(* IEC 61131-3 sources: Industry-PLC-LLM/data/PLCBEAD_repo/PLCBEAD_PLCEmbed-main/PLC-BEAD/Source/OpenPLCv2 (part 12) *)

(* ---- RES_NI.ST ---- *)
FUNCTION RES_NI:REAL

	VAR_INPUT
		T :	REAL;
		R0 :	REAL;
	END_VAR

	VAR
		T2 :	REAL;
	END_VAR

	T2 := T*T;
	Res_NI := R0 + 0.5485*T + 0.665E-3*T2 + 2.805E-9*T2*T2;

END_FUNCTION

PROGRAM program0

	VAR
		T :	REAL;
		R0 :	REAL;

		OUT :	REAL;
	END_VAR
	OUT := RES_NI(T, R0);

END_PROGRAM

CONFIGURATION Config0

	RESOURCE Res0 ON PLC
		TASK task0(INTERVAL := T#20ms,PRIORITY := 0);
		PROGRAM instance0 WITH task0 : program0;
	END_RESOURCE

END_CONFIGURATION

(* ---- RES_NTC.ST ---- *)
FUNCTION RES_NTC:REAL

	VAR_INPUT
		T :	REAL;
		RN :	REAL;
		B :	REAL;
	END_VAR

	RES_NTC := RN * EXP(B * (1.0 / (T+273.15) - 0.00335401643468053));

END_FUNCTION

PROGRAM program0

	VAR
		T :	REAL;
		RN :	REAL;
		B :	REAL;

		OUT :	REAL;
	END_VAR
		OUT := RES_NTC(T, RN, B);

END_PROGRAM

CONFIGURATION Config0

	RESOURCE Res0 ON PLC
		TASK task0(INTERVAL := T#20ms,PRIORITY := 0);
		PROGRAM instance0 WITH task0 : program0;
	END_RESOURCE

END_CONFIGURATION

(* ---- RES_PT.ST ---- *)
FUNCTION RES_PT:REAL
	VAR_INPUT
		T :	REAL;
		R0 :	REAL;
	END_VAR

	VAR
		T2 :	REAL;
	END_VAR

	T2 := T * T;

	IF T >= 0.0 THEN
		RES_PT := R0 * ( 1.0 + 3.90802E-3 * T + -5.802E-7 * T2);
	ELSE
		RES_PT := R0 * ( 1.0 + 3.90802E-3 * T + -5.802E-7 * T2 + -4.27350E-12 * (T - 100.0) * T2 * T);
	END_IF;

END_FUNCTION

PROGRAM program0
  	VAR
		T :	REAL;
		R0 : REAL;
		CEIL5_OUT : REAL;
  	END_VAR

  	CEIL5_OUT := RES_PT(T, R0);
END_PROGRAM

CONFIGURATION Config0
	RESOURCE Res0 ON PLC
		TASK task0(INTERVAL := T#20ms,PRIORITY := 0);
		PROGRAM instance0 WITH task0 : program0;
	END_RESOURCE
END_CONFIGURATION

(* ---- RES_SI.ST ---- *)
FUNCTION RES_SI:REAL

	VAR_INPUT
		T :	REAL;
		_RS :	REAL;
		TS :	REAL;
	END_VAR

	VAR
		TX :	REAL;
	END_VAR

	TX := T - TS;
	RES_SI := _RS * ( 1.0 + 7.64E-3 * TX + 1.66E-5 * TX * TX);

END_FUNCTION

PROGRAM program0

	VAR
		T :	REAL;
		_RS :	REAL;
		TS :	REAL;

		OUT :	REAL;
	END_VAR
		OUT := RES_SI(T, _RS, TS);

END_PROGRAM

CONFIGURATION Config0

	RESOURCE Res0 ON PLC
		TASK task0(INTERVAL := T#20ms,PRIORITY := 0);
		PROGRAM instance0 WITH task0 : program0;
	END_RESOURCE

END_CONFIGURATION

(* ---- REVERSE.ST ---- *)
FUNCTION REVERSE:BYTE
VAR_INPUT
	IN :	BYTE;
END_VAR

reverse := SHL(in,7) OR SHR(in,7) OR (ROR(in,3) AND BYTE#2#01000100) OR (ROL(in,3) AND BYTE#2#00100010)
	OR (SHL(in,1) AND BYTE#2#00010000) OR (SHR(in,1) AND BYTE#2#00001000);

END_FUNCTION

PROGRAM program0
  VAR
    LocalVar0 : BYTE;
	LocalOUT  : BYTE;
  END_VAR
  	LocalOUT := REVERSE(LocalVar0);
END_PROGRAM

CONFIGURATION Config0
  RESOURCE Res0 ON PLC
    TASK task0(INTERVAL := T#20ms,PRIORITY := 0);
    PROGRAM instance0 WITH task0 : program0;
  END_RESOURCE
END_CONFIGURATION

(* ---- RND.ST ---- *)
FUNCTION CEIL:INT

	VAR_INPUT
		X :	REAL;
	END_VAR

	CEIL := REAL_TO_INT(x);
	IF INT_TO_REAL(CEIL) < X THEN
			CEIL := CEIL + 1;
	END_IF;

END_FUNCTION

FUNCTION BIT_OF_DWORD : BOOL

	VAR_INPUT
		IN : DWORD;
		N : INT;
	END_VAR

	BIT_OF_DWORD := (SHR(in,N) AND 16#00000001) > 0;

END_FUNCTION

FUNCTION EXPN:REAL

	VAR_INPUT
		X :	REAL;
		N :	INT;
	END_VAR

	VAR
		N_word :	WORD;
		X_tmp :	REAL;
		sign :	BOOL;
	END_VAR

	N_word := INT_TO_WORD(N);
	X_tmp := X;
	sign := BIT_OF_DWORD(WORD_TO_DWORD(N_word),15);
	N_word := INT_TO_WORD(ABS(N));
	IF BIT_OF_DWORD(WORD_TO_DWORD(N_word),0) THEN expn := X_tmp; ELSE expn := 1.0; END_IF;    (* N_word.X0 *)
	N_word := SHR(N_word,1);
	WHILE N_word > WORD#0 DO
		X_tmp := X_tmp * X_tmp;
		IF BIT_OF_DWORD(WORD_TO_DWORD(N_word),0) THEN expn := expn * X_tmp; END_IF;       (* N_word.X0 *)
		N_word := SHR(N_word,1);
	END_WHILE;
	IF sign THEN EXPN := 1.0 / EXPN; END_IF;

END_FUNCTION

FUNCTION _REAL_TO_DINT:DINT
	VAR_INPUT
		X :	REAL;
	END_VAR

	IF REAL_TO_DINT(0.5) = DINT#1 THEN
		_REAL_TO_DINT := REAL_TO_DINT(x);
		RETURN;
	END_IF;

	IF X > 0.0 THEN
		_REAL_TO_DINT := REAL_TO_DINT(x+0.5);
	ELSIF X < 0.0 THEN
		_REAL_TO_DINT := REAL_TO_DINT(x-0.5);
	ELSE
		_REAL_TO_DINT := DINT#0;
	END_IF;
END_FUNCTION

FUNCTION RND:REAL

	VAR_INPUT
		X :	REAL;
		N :	INT;
	END_VAR

	VAR
		M :	REAL;
	END_VAR

	IF X = 0.0 THEN
		RND := 0.0;
	ELSE
		M := EXPN(10.0,N - CEIL(LOG(ABS(X))));
		RND := DINT_TO_REAL(_REAL_TO_DINT(X * M)) / M;
	END_IF;

END_FUNCTION

PROGRAM program0
	VAR
		IN : REAL;
		N :	INT;
		X :	REAL;
	END_VAR
		X := RND(IN, N);
END_PROGRAM

CONFIGURATION Config0

	RESOURCE Res0 ON PLC
		TASK task0(INTERVAL := T#20ms,PRIORITY := 0);
		PROGRAM instance0 WITH task0 : program0;
	END_RESOURCE

END_CONFIGURATION

(* ---- ROUND.ST ---- *)
FUNCTION _REAL_TO_DINT:DINT
	VAR_INPUT
		X :	REAL;
	END_VAR

	IF REAL_TO_DINT(0.5) = DINT#1 THEN
		_REAL_TO_DINT := REAL_TO_DINT(x);
		RETURN;
	END_IF;

	IF X > 0.0 THEN
		_REAL_TO_DINT := REAL_TO_DINT(x+0.5);
	ELSIF X < 0.0 THEN
		_REAL_TO_DINT := REAL_TO_DINT(x-0.5);
	ELSE
		_REAL_TO_DINT := DINT#0;
	END_IF;
END_FUNCTION

FUNCTION ROUND:REAL

	VAR_INPUT
		IN :	REAL;
		N :	INT;
	END_VAR

	VAR
		X :	REAL;
	END_VAR

	IF N < 4 THEN
		IF N < 2 THEN
			IF N = 0 THEN X := 1.0; ELSE X := 10.0; END_IF;
		ELSE
			IF N = 2 THEN X := 100.0; ELSE X := 1000.0; END_IF;
		END_IF;
	ELSE
		IF N < 6 THEN
			IF N = 4 THEN X := 10000.0; ELSE X := 100000.0; END_IF;
		ELSE
			IF N = 6 THEN X := 1000000.0; ELSE X := 10000000.0; END_IF;
		END_IF;
	END_IF;

	ROUND := DINT_TO_REAL(_REAL_TO_DINT(in * X)) / X;

END_FUNCTION

PROGRAM program0
	VAR
		IN : REAL;
		N :	INT;
		X :	REAL;
	END_VAR
		X := ROUND(IN, N);
END_PROGRAM

CONFIGURATION Config0

	RESOURCE Res0 ON PLC
		TASK task0(INTERVAL := T#20ms,PRIORITY := 0);
		PROGRAM instance0 WITH task0 : program0;
	END_RESOURCE

END_CONFIGURATION

(* ---- SCALE.ST ---- *)
FUNCTION SCALE:REAL

	VAR_INPUT
		X :	REAL;
		K :	REAL;
		O :	REAL;
		MX :	REAL;
		MN :	REAL;
	END_VAR

	SCALE := LIMIT(MN, X * K + O, MX);

END_FUNCTION

PROGRAM program0
  VAR
    X :	REAL;
	K :	REAL;
	O :	REAL;
	MX :	REAL;
	MN :	REAL;
    CEIL5_OUT : REAL;
  END_VAR

  CEIL5_OUT := SCALE(X, K, O, MX, MN);
END_PROGRAM

CONFIGURATION Config0

  RESOURCE Res0 ON PLC
    TASK task0(INTERVAL := T#20ms,PRIORITY := 0);
    PROGRAM instance0 WITH task0 : program0;
  END_RESOURCE
END_CONFIGURATION

(* ---- SCALE_B.ST ---- *)
FUNCTION _BYTE_TO_REAL:REAL
	VAR_INPUT
		IN :	BYTE;
	END_VAR

	_BYTE_TO_REAL := USINT_TO_REAL(BYTE_TO_USINT(IN));
END_FUNCTION

FUNCTION SCALE_B:REAL

	VAR_INPUT
		X :	BYTE;
		I_LO :	BYTE;
		I_HI :	BYTE;
		O_LO :	REAL;
		O_HI :	REAL;
	END_VAR

	IF I_HI = I_LO THEN
		SCALE_B := O_LO;
	ELSE
		SCALE_B := (O_HI - O_LO) / USINT_TO_REAL(BYTE_TO_USINT(I_HI) - BYTE_TO_USINT(I_LO)) * _BYTE_TO_REAL(LIMIT(I_LO,X,I_HI));
	END_IF;

END_FUNCTION

PROGRAM program0
  VAR
	X :	BYTE;
	I_LO :	BYTE;
	I_HI :	BYTE;
	O_LO :	REAL;
	O_HI :	REAL;
	CEIL5_OUT : REAL;
  END_VAR

  CEIL5_OUT := SCALE_B(X, I_LO, I_HI, O_LO, O_HI);

END_PROGRAM

CONFIGURATION Config0

  RESOURCE Res0 ON PLC
    TASK task0(INTERVAL := T#20ms,PRIORITY := 0);
    PROGRAM instance0 WITH task0 : program0;
  END_RESOURCE
END_CONFIGURATION

(* ---- SCALE_B2.ST ---- *)
FUNCTION _BYTE_TO_REAL:REAL
	VAR_INPUT
		IN :	BYTE;
	END_VAR

	_BYTE_TO_REAL := USINT_TO_REAL(BYTE_TO_USINT(IN));
END_FUNCTION

FUNCTION SCALE_B2:REAL
	VAR_INPUT
		IN1 :	BYTE;
		IN2 :	BYTE;
		K :	REAL;
		O :	REAL;
		IN1_MIN :	REAL;
		IN1_MAX :	REAL;
		IN2_MIN :	REAL;
		IN2_MAX :	REAL;
	END_VAR

	SCALE_B2 := 	(((in1_max - in1_min)* _BYTE_TO_REAL(in1) + (in2_max - in2_min)* _BYTE_TO_REAL(in2)) * 0.003921569 + in1_min + in2_min) * K + O;

END_FUNCTION

PROGRAM program0
  VAR
	IN1 :	BYTE;
	IN2 :	BYTE;
	K :	REAL;
	O :	REAL;
	IN1_MIN :	REAL;
	IN1_MAX :	REAL;
	IN2_MIN :	REAL;
	IN2_MAX :	REAL;
	CEIL5_OUT : REAL;
  END_VAR

  CEIL5_OUT := SCALE_B2(IN1, IN2, K, O, IN1_MIN, IN1_MAX, IN2_MIN, IN2_MAX);

END_PROGRAM

CONFIGURATION Config0

  RESOURCE Res0 ON PLC
    TASK task0(INTERVAL := T#20ms,PRIORITY := 0);
    PROGRAM instance0 WITH task0 : program0;
  END_RESOURCE
END_CONFIGURATION

(* ---- SCALE_B4.ST ---- *)
FUNCTION _BYTE_TO_REAL:REAL
	VAR_INPUT
		IN :	BYTE;
	END_VAR

	_BYTE_TO_REAL := USINT_TO_REAL(BYTE_TO_USINT(IN));
END_FUNCTION

FUNCTION SCALE_B4:REAL

	VAR_INPUT
		IN1 :	BYTE;
		IN2 :	BYTE;
		IN3 :	BYTE;
		IN4 :	BYTE;
		K :	REAL;
		O :	REAL;
		IN1_MIN :	REAL;
		IN1_MAX :	REAL;
		IN2_MIN :	REAL;
		IN2_MAX :	REAL;
		IN3_MIN :	REAL;
		IN3_MAX :	REAL;
		IN4_MIN :	REAL;
		IN4_MAX :	REAL;
	END_VAR

	SCALE_B4 := 	(((in1_max - in1_min)* _BYTE_TO_REAL(in1) + (in2_max - in2_min)* _BYTE_TO_REAL(in2) + (in3_max - in3_min)* _BYTE_TO_REAL(in3) + (in4_max - in4_min)* _BYTE_TO_REAL(in4))* 0.003921569 + in1_min + in2_min + in3_min + in4_min) * K + O;

END_FUNCTION

PROGRAM program0
  VAR
	IN1 :	BYTE;
	IN2 :	BYTE;
	IN3 :	BYTE;
	IN4 :	BYTE;
	K :	REAL;
	O :	REAL;
	IN1_MIN :	REAL;
	IN1_MAX :	REAL;
	IN2_MIN :	REAL;
	IN2_MAX :	REAL;
	IN3_MIN :	REAL;
	IN3_MAX :	REAL;
	IN4_MIN :	REAL;
	IN4_MAX :	REAL;
	CEIL5_OUT : REAL;
  END_VAR

  CEIL5_OUT := SCALE_B4(IN1, IN2, IN3, IN4, K, O, IN1_MIN, IN1_MAX, IN2_MIN, IN2_MAX, IN3_MIN, IN3_MAX, IN4_MIN, IN4_MAX);

END_PROGRAM

CONFIGURATION Config0

  RESOURCE Res0 ON PLC
    TASK task0(INTERVAL := T#20ms,PRIORITY := 0);
    PROGRAM instance0 WITH task0 : program0;
  END_RESOURCE
END_CONFIGURATION

(* ---- SCALE_B8.ST ---- *)
FUNCTION _BYTE_TO_REAL:REAL
	VAR_INPUT
		IN :	BYTE;
	END_VAR

	_BYTE_TO_REAL := USINT_TO_REAL(BYTE_TO_USINT(IN));
END_FUNCTION

FUNCTION SCALE_B8:REAL
	VAR_INPUT
		IN1 :	BYTE;
		IN2 :	BYTE;
		IN3 :	BYTE;
		IN4 :	BYTE;
		IN5 :	BYTE;
		IN6 :	BYTE;
		IN7 :	BYTE;
		IN8 :	BYTE;
		K :	REAL;
		O :	REAL;
		IN1_MIN :	REAL;
		IN1_MAX :	REAL;
		IN2_MIN :	REAL;
		IN2_MAX :	REAL;
		IN3_MIN :	REAL;
		IN3_MAX :	REAL;
		IN4_MIN :	REAL;
		IN4_MAX :	REAL;
		IN5_MIN :	REAL;
		IN5_MAX :	REAL;
		IN6_MIN :	REAL;
		IN6_MAX :	REAL;
		IN7_MIN :	REAL;
		IN7_MAX :	REAL;
		IN8_MIN :	REAL;
		IN8_MAX :	REAL;
	END_VAR

	SCALE_B8 := 	(((in1_max - in1_min)* _BYTE_TO_REAL(in1) + (in2_max - in2_min)* _BYTE_TO_REAL(in2) + (in3_max - in3_min)* _BYTE_TO_REAL(in3) + (in4_max - in4_min)* _BYTE_TO_REAL(in4) +
					(in5_max - in5_min)* _BYTE_TO_REAL(in5) + (in6_max - in6_min)* _BYTE_TO_REAL(in6) + (in7_max - in7_min)* _BYTE_TO_REAL(in7) + (in8_max - in8_min)* _BYTE_TO_REAL(in8)) * 0.003921569
					+ in1_min + in2_min + in3_min + in4_min + in5_min + in6_min + in7_min + in8_min) * K + O;

END_FUNCTION

PROGRAM program0
  	VAR
		IN1 :	BYTE;
		IN2 :	BYTE;
		IN3 :	BYTE;
		IN4 :	BYTE;
		IN5 :	BYTE;
		IN6 :	BYTE;
		IN7 :	BYTE;
		IN8 :	BYTE;
		K :	REAL;
		O :	REAL;
		IN1_MIN :	REAL;
		IN1_MAX :	REAL;
		IN2_MIN :	REAL;
		IN2_MAX :	REAL;
		IN3_MIN :	REAL;
		IN3_MAX :	REAL;
		IN4_MIN :	REAL;
		IN4_MAX :	REAL;
		IN5_MIN :	REAL;
		IN5_MAX :	REAL;
		IN6_MIN :	REAL;
		IN6_MAX :	REAL;
		IN7_MIN :	REAL;
		IN7_MAX :	REAL;
		IN8_MIN :	REAL;
		IN8_MAX :	REAL;
		CEIL5_OUT : REAL;
  	END_VAR

  	CEIL5_OUT := SCALE_B8(IN1, IN2, IN3, IN4, IN5, IN6, IN7, IN8, K, O, IN1_MIN, IN1_MAX, IN2_MIN, IN2_MAX, IN3_MIN, IN3_MAX, IN4_MIN, IN4_MAX, IN5_MIN, IN5_MAX, IN6_MIN, IN6_MAX, IN7_MIN, IN7_MAX, IN8_MIN, IN8_MAX);

	END_PROGRAM

CONFIGURATION Config0

	RESOURCE Res0 ON PLC
		TASK task0(INTERVAL := T#20ms,PRIORITY := 0);
		PROGRAM instance0 WITH task0 : program0;
	END_RESOURCE

END_CONFIGURATION

(* ---- SCALE_D.ST ---- *)
FUNCTION SCALE_D:REAL
	VAR_INPUT
		X :	DWORD;
		I_LO :	DWORD;
		I_HI :	DWORD;
		O_LO :	REAL;
		O_HI :	REAL;
	END_VAR
	IF I_HI = I_LO THEN
		SCALE_D := O_LO;
	ELSE
		SCALE_D := (O_HI - O_LO) / UDINT_TO_REAL(DWORD_TO_UDINT(I_HI) - DWORD_TO_UDINT(I_LO)) * UDINT_TO_REAL(LIMIT(DWORD_TO_UDINT(I_LO),DWORD_TO_UDINT(X),DWORD_TO_UDINT(I_HI)) - DWORD_TO_UDINT(I_LO)) + O_LO;
	END_IF;
END_FUNCTION

PROGRAM program0
  VAR
		X :	DWORD;
		I_LO :	DWORD;
		I_HI :	DWORD;
		O_LO :	REAL;
		O_HI :	REAL;
		CEIL5_OUT : REAL;
  END_VAR

  CEIL5_OUT := SCALE_D(X, I_LO, I_HI, O_LO, O_HI);
END_PROGRAM

CONFIGURATION Config0

  RESOURCE Res0 ON PLC
    TASK task0(INTERVAL := T#20ms,PRIORITY := 0);
    PROGRAM instance0 WITH task0 : program0;
  END_RESOURCE
END_CONFIGURATION

(* ---- SCALE_R.ST ---- *)
FUNCTION SCALE_R:REAL
	VAR_INPUT
		X :	REAL;
		I_LO :	REAL;
		I_HI :	REAL;
		O_LO :	REAL;
		O_HI :	REAL;
	END_VAR

	IF I_LO = I_HI THEN
		SCALE_R := O_LO;
	ELSE
		SCALE_R := (O_HI - O_LO) / (I_HI - I_LO) * (LIMIT(I_LO, X, I_HI) - I_LO) + O_LO;
	END_IF;

END_FUNCTION

PROGRAM program0

  	VAR
		X :	REAL;
		I_LO :	REAL;
		I_HI :	REAL;
		O_LO :	REAL;
		O_HI :	REAL;
		CEIL5_OUT : REAL;
  	END_VAR

  	CEIL5_OUT := SCALE_R(X, I_LO, I_HI, O_LO, O_HI);
END_PROGRAM

CONFIGURATION Config0

	RESOURCE Res0 ON PLC
		TASK task0(INTERVAL := T#20ms,PRIORITY := 0);
		PROGRAM instance0 WITH task0 : program0;
	END_RESOURCE

END_CONFIGURATION

(* ---- SCALE_X2.ST ---- *)
FUNCTION SCALE_X2:REAL
	VAR_INPUT
		IN1 :	BOOL;
		IN2 :	BOOL;
		K :	REAL;
		O :	REAL;
		IN1_MIN :	REAL;(*Standard = 0*)
		IN1_MAX :	REAL;(*Standard = 1000*)
		IN2_MIN :	REAL;(*Standard = 0*)
		IN2_MAX :	REAL;(*Standard = 1000*)
	END_VAR

	SCALE_X2 := (SEL(IN1,IN1_MIN, IN1_MAX)+ SEL(IN2,IN2_MIN, IN2_MAX))* k + o;

END_FUNCTION

PROGRAM program0

  	VAR
		IN1 :	BOOL;
		IN2 :	BOOL;
		K :	REAL;
		O :	REAL;
		IN1_MIN :	REAL;(*Standard = 0*)
		IN1_MAX :	REAL;(*Standard = 1000*)
		IN2_MIN :	REAL;(*Standard = 0*)
		IN2_MAX :	REAL;(*Standard = 1000*)
		CEIL5_OUT : REAL;
  	END_VAR

  	CEIL5_OUT := SCALE_X2(IN1, IN2, K, O, IN1_MIN, IN1_MAX, IN2_MIN, IN2_MAX);
END_PROGRAM

CONFIGURATION Config0

	RESOURCE Res0 ON PLC
		TASK task0(INTERVAL := T#20ms,PRIORITY := 0);
		PROGRAM instance0 WITH task0 : program0;
	END_RESOURCE

END_CONFIGURATION

(* ---- SCALE_X4.ST ---- *)
FUNCTION SCALE_X4:REAL
	VAR_INPUT
		IN1 :	BOOL;
		IN2 :	BOOL;
		IN3 :	BOOL;
		IN4 :	BOOL;
		K :	REAL;
		O :	REAL;
		IN1_MIN :	REAL;
		IN1_MAX :	REAL;
		IN2_MIN :	REAL;
		IN2_MAX :	REAL;
		IN3_MIN :	REAL;
		IN3_MAX :	REAL;
		IN4_MIN :	REAL;
		IN4_MAX :	REAL;
	END_VAR
	IF NOT in1 THEN scale_X4 := in1_min; ELSE scale_X4 := in1_max; END_IF;
	IF NOT in2 THEN scale_x4 := scale_x4 + in2_min; ELSE scale_x4 := scale_x4 + in2_max; END_IF;
	IF NOT in3 THEN scale_x4 := scale_x4 + in3_min; ELSE scale_x4 := scale_x4 + in3_max; END_IF;
	IF NOT in4 THEN scale_x4 := scale_x4 + in4_min; ELSE scale_x4 := scale_x4 + in4_max; END_IF;
	scale_X4 := scale_X4 * k + O;
	END_FUNCTION

PROGRAM program0

  	VAR
		IN1 :	BOOL;
		IN2 :	BOOL;
		IN3 :	BOOL;
		IN4 :	BOOL;
		K :	REAL;
		O :	REAL;
		IN1_MIN :	REAL;
		IN1_MAX :	REAL;
		IN2_MIN :	REAL;
		IN2_MAX :	REAL;
		IN3_MIN :	REAL;
		IN3_MAX :	REAL;
		IN4_MIN :	REAL;
		IN4_MAX :	REAL;
		CEIL5_OUT : REAL;
  	END_VAR

  	CEIL5_OUT := SCALE_X4(IN1, IN2, IN3, IN4, K, O, IN1_MIN, IN1_MAX, IN2_MIN, IN2_MAX, IN3_MIN, IN3_MAX, IN4_MIN, IN4_MAX);
END_PROGRAM

CONFIGURATION Config0

	RESOURCE Res0 ON PLC
		TASK task0(INTERVAL := T#20ms,PRIORITY := 0);
		PROGRAM instance0 WITH task0 : program0;
	END_RESOURCE

END_CONFIGURATION

(* ---- SCALE_X8.ST ---- *)
FUNCTION SCALE_X8:REAL

	VAR_INPUT
		IN1 :	BOOL;
		IN2 :	BOOL;
		IN3 :	BOOL;
		IN4 :	BOOL;
		IN5 :	BOOL;
		IN6 :	BOOL;
		IN7 :	BOOL;
		IN8 :	BOOL;
		K :	REAL;
		O :	REAL;
		IN1_MIN :	REAL;
		IN1_MAX :	REAL;
		IN2_MIN :	REAL;
		IN2_MAX :	REAL;
		IN3_MIN :	REAL;
		IN3_MAX :	REAL;
		IN4_MIN :	REAL;
		IN4_MAX :	REAL;
		IN5_MIN :	REAL;
		IN5_MAX :	REAL;
		IN6_MIN :	REAL;
		IN6_MAX :	REAL;
		IN7_MIN :	REAL;
		IN7_MAX :	REAL;
		IN8_MIN :	REAL;
		IN8_MAX :	REAL;
	END_VAR

	SCALE_X8 := (SEL(IN1,IN1_MIN, IN1_MAX)+ SEL(IN2,IN2_MIN, IN2_MAX)+SEL(IN3,IN3_MIN, IN3_MAX)+ SEL(IN4,IN4_MIN, IN4_MAX)
					+SEL(IN5,IN5_MIN, IN5_MAX)+ SEL(IN6,IN6_MIN, IN6_MAX)+SEL(IN7,IN7_MIN, IN7_MAX)+ SEL(IN8,IN8_MIN, IN8_MAX))*k + o;

END_FUNCTION

PROGRAM program0

  	VAR
		IN1 :	BOOL;
		IN2 :	BOOL;
		IN3 :	BOOL;
		IN4 :	BOOL;
		IN5 :	BOOL;
		IN6 :	BOOL;
		IN7 :	BOOL;
		IN8 :	BOOL;
		K :	REAL;
		O :	REAL;
		IN1_MIN :	REAL;
		IN1_MAX :	REAL;
		IN2_MIN :	REAL;
		IN2_MAX :	REAL;
		IN3_MIN :	REAL;
		IN3_MAX :	REAL;
		IN4_MIN :	REAL;
		IN4_MAX :	REAL;
		IN5_MIN :	REAL;
		IN5_MAX :	REAL;
		IN6_MIN :	REAL;
		IN6_MAX :	REAL;
		IN7_MIN :	REAL;
		IN7_MAX :	REAL;
		IN8_MIN :	REAL;
		IN8_MAX :	REAL;
		CEIL5_OUT : REAL;
  	END_VAR

  	CEIL5_OUT := SCALE_X8(IN1, IN2, IN3, IN4, IN5, IN6, IN7, IN8, K, O, IN1_MIN, IN1_MAX, IN2_MIN, IN2_MAX, IN3_MIN, IN3_MAX, IN4_MIN, IN4_MAX, IN5_MIN, IN5_MAX, IN6_MIN, IN6_MAX, IN7_MIN, IN7_MAX, IN8_MIN, IN8_MAX);
END_PROGRAM

CONFIGURATION Config0

	RESOURCE Res0 ON PLC
		TASK task0(INTERVAL := T#20ms,PRIORITY := 0);
		PROGRAM instance0 WITH task0 : program0;
	END_RESOURCE

END_CONFIGURATION

(* ---- SDD.ST ---- *)
FUNCTION SDD:REAL

	VAR_INPUT
		T :	REAL;
		ICE :	BOOL;
	END_VAR

	IF ice THEN
		SDD := 611.153 * EXP(22.4433 * T / (272.186 + T));
	ELSE
		SDD := 611.213 * EXP(17.5043 * T / (241.2 + T));
	END_IF;

END_FUNCTION

PROGRAM program0
  VAR
    T :	REAL;
	ICE :	BOOL;
    CEIL5_OUT : REAL;
  END_VAR

  CEIL5_OUT := SDD(T, ICE);
END_PROGRAM

CONFIGURATION Config0

  RESOURCE Res0 ON PLC
    TASK task0(INTERVAL := T#20ms,PRIORITY := 0);
    PROGRAM instance0 WITH task0 : program0;
  END_RESOURCE
END_CONFIGURATION

(* ---- SDD_NH3.ST ---- *)
FUNCTION SDD_NH3:REAL

	VAR_INPUT
		T :	REAL;
	END_VAR

	IF T < -33.65 THEN
		SDD_NH3 := EXP(7.3396511649 - ( 1166.7498002 / ( T + 192.37 )));
	ELSE
		SDD_NH3 := EXP(11.210964456 - ( 2564.9140075 / ( T + 262.741 )));
	END_IF;

END_FUNCTION

PROGRAM program0
  VAR
    T :	REAL;
    CEIL5_OUT : REAL;
  END_VAR

  CEIL5_OUT := SDD_NH3(T);
END_PROGRAM

CONFIGURATION Config0

  RESOURCE Res0 ON PLC
    TASK task0(INTERVAL := T#20ms,PRIORITY := 0);
    PROGRAM instance0 WITH task0 : program0;
  END_RESOURCE
END_CONFIGURATION

(* ---- SDT_NH3.ST ---- *)
FUNCTION SDT_NH3:REAL

	VAR_INPUT
		P :	REAL;
	END_VAR

	IF P < 1.0E-3 THEN
		SDT_NH3 := -110.0;
	ELSIF P < 1.0 THEN
		SDT_NH3 := 506.713 / (3.18757 - LOG(P)) - 192.37 ;
	ELSE
		SDT_NH3 := 1113.928 / (4.86886 - LOG(P)) - 262.71 ;
	END_IF;

END_FUNCTION

PROGRAM program0
  VAR
    P :	REAL;
    CEIL5_OUT : REAL;
  END_VAR

  CEIL5_OUT := SDT_NH3(P);
END_PROGRAM

CONFIGURATION Config0

  RESOURCE Res0 ON PLC
    TASK task0(INTERVAL := T#20ms,PRIORITY := 0);
    PROGRAM instance0 WITH task0 : program0;
  END_RESOURCE
END_CONFIGURATION

(* ---- SECOND.ST ---- *)
FUNCTION SECOND:REAL

	VAR_INPUT
		ITOD :	UDINT;
	END_VAR

	second := UDINT_TO_REAL(itod MOD UDINT#60000) / REAL#1000.00;

END_FUNCTION

PROGRAM program0
  VAR
    ITOD :	UDINT;
    CEIL5_OUT : REAL;
  END_VAR

  CEIL5_OUT := SECOND(ITOD);
END_PROGRAM

CONFIGURATION Config0

	RESOURCE Res0 ON PLC
		TASK task0(INTERVAL := T#20ms,PRIORITY := 0);
		PROGRAM instance0 WITH task0 : program0;
	END_RESOURCE

END_CONFIGURATION

(* ---- SECOND_OF_DT.ST ---- *)
FUNCTION SECOND_OF_DT:INT

	VAR_INPUT
		XDT :	UDINT;
	END_VAR

	SECOND_OF_DT := UDINT_TO_INT(XDT MOD UDINT#60);
END_FUNCTION

PROGRAM program0
  VAR
    LocalVar0 : UDINT;
	LocalOUT  : INT;
  END_VAR
  	LocalOUT := SECOND_OF_DT(LocalVar0);
END_PROGRAM

CONFIGURATION Config0
  RESOURCE Res0 ON PLC
    TASK task0(INTERVAL := T#20ms,PRIORITY := 0);
    PROGRAM instance0 WITH task0 : program0;
  END_RESOURCE
END_CONFIGURATION

(* ---- SECOND_TO_TIME.ST ---- *)
FUNCTION _REAL_TO_UDINT:UDINT
	VAR_INPUT
		X :	REAL;
	END_VAR

	IF REAL_TO_UDINT(0.5) = UDINT#1 THEN
		_REAL_TO_UDINT := REAL_TO_UDINT(x);
	ELSIF X > 0.0 THEN
		_REAL_TO_UDINT := REAL_TO_UDINT(x+0.5);
	ELSIF X < 0.0 THEN
		_REAL_TO_UDINT := REAL_TO_UDINT(x-0.5);
	ELSE
		_REAL_TO_UDINT := UDINT#0;
	END_IF;
END_FUNCTION

FUNCTION SECOND_TO_TIME:TIME

	VAR_INPUT
		IN :	REAL;
	END_VAR

	second_to_time := UDINT_TO_TIME(_REAL_TO_UDINT(IN * 1000.0));

END_FUNCTION

PROGRAM program0

	VAR
		IN :	REAL;
		CEIL5_OUT : TIME;
	END_VAR

	CEIL5_OUT := SECOND_TO_TIME(IN);

END_PROGRAM

CONFIGURATION Config0

	RESOURCE Res0 ON PLC
		TASK task0(INTERVAL := T#20ms,PRIORITY := 0);
		PROGRAM instance0 WITH task0 : program0;
	END_RESOURCE

END_CONFIGURATION

(* ---- SENSOR_INT.ST ---- *)
FUNCTION SENSOR_INT:REAL

	VAR_INPUT
		VOLTAGE :	REAL;
		CURRENT :	REAL;
		RP :	REAL;
		_RS :	REAL;
	END_VAR

	VAR
		RG :	REAL;
	END_VAR

	IF current <> 0.0 THEN
		RG := voltage / current;
		SENSOR_INT := RP * ( RG - _RS) / ( RP + _RS - RG);
	END_IF;

END_FUNCTION

PROGRAM program0

	VAR
		VOLTAGE :	REAL;
		CURRENT :	REAL;
		RP :	REAL;
		_RS :	REAL;
		CEIL5_OUT : REAL;
	END_VAR

	CEIL5_OUT := SENSOR_INT(VOLTAGE, CURRENT, RP, _RS);

END_PROGRAM

CONFIGURATION Config0

	RESOURCE Res0 ON PLC
		TASK task0(INTERVAL := T#20ms,PRIORITY := 0);
		PROGRAM instance0 WITH task0 : program0;
	END_RESOURCE

END_CONFIGURATION

(* ---- SET_DATE.ST ---- *)
FUNCTION _INT_TO_UDINT:UDINT
	VAR_INPUT
		IN :	INT;
	END_VAR

	_INT_TO_UDINT := DINT_TO_UDINT(INT_TO_DINT(IN));
END_FUNCTION

FUNCTION SET_DATE:UDINT

	VAR_INPUT
		YEAR :	INT;
		MONTH :	INT;
		DAY :	INT;
	END_VAR

	VAR
		count :	INT;
	END_VAR

	IF month > 2 THEN
		count := (month - 1) * 30;
		IF month > 7 THEN
			count := count + DWORD_TO_INT(SHR(DINT_TO_DWORD(INT_TO_DINT(month) - INT_TO_DINT(3)),1));
		ELSE
			count := count + DWORD_TO_INT(SHR(DINT_TO_DWORD(INT_TO_DINT(month) - INT_TO_DINT(4)),1));
		END_IF;
		IF SHL(INT_TO_WORD(year),14) = WORD#0 THEN
			count := count + 1;
		END_IF;
	ELSE
		count := (month - 1) * 31;
	END_IF;
	SET_DATE := (_INT_TO_UDINT(count + day - 1) + DWORD_TO_UDINT(SHR(UDINT_TO_DWORD(_INT_TO_UDINT(year) * UDINT#1461 - UDINT#2878169), 2))) * UDINT#86400;

END_FUNCTION

PROGRAM program0
  VAR
	YEAR :	INT;
	MONTH :	INT;
	DAY :	INT;
    CEIL5_OUT : UDINT;
  END_VAR

  CEIL5_OUT := SET_DATE(YEAR, MONTH, DAY);
END_PROGRAM

CONFIGURATION Config0

  RESOURCE Res0 ON PLC
    TASK task0(INTERVAL := T#20ms,PRIORITY := 0);
    PROGRAM instance0 WITH task0 : program0;
  END_RESOURCE
END_CONFIGURATION

(* ---- SET_DT.ST ---- *)
FUNCTION _INT_TO_UDINT:UDINT
	VAR_INPUT
		IN :	INT;
	END_VAR

	_INT_TO_UDINT := DINT_TO_UDINT(INT_TO_DINT(IN));
END_FUNCTION

FUNCTION SET_DATE:UDINT

	VAR_INPUT
		YEAR :	INT;
		MONTH :	INT;
		DAY :	INT;
	END_VAR

	VAR
		count :	INT;
	END_VAR

	IF month > 2 THEN
		count := (month - 1) * 30;
		IF month > 7 THEN
			count := count + DWORD_TO_INT(SHR(DINT_TO_DWORD(INT_TO_DINT(month) - INT_TO_DINT(3)),1));
		ELSE
			count := count + DWORD_TO_INT(SHR(DINT_TO_DWORD(INT_TO_DINT(month) - INT_TO_DINT(4)),1));
		END_IF;
		IF SHL(INT_TO_WORD(year),14) = WORD#0 THEN
			count := count + 1;
		END_IF;
	ELSE
		count := (month - 1) * 31;
	END_IF;
	SET_DATE := (_INT_TO_UDINT(count + day - 1) + DWORD_TO_UDINT(SHR(UDINT_TO_DWORD(_INT_TO_UDINT(year) * UDINT#1461 - UDINT#2878169), 2))) * UDINT#86400;

END_FUNCTION

FUNCTION SET_DT:UDINT
	VAR_INPUT
		YEAR :	INT;
		MONTH :	INT;
		DAY :	INT;
		HOUR :	INT;
		MINUTE :	INT;
		SECOND :	INT;
	END_VAR

	SET_DT := SET_DATE(YEAR, MONTH, DAY) + _INT_TO_UDINT(SECOND) + _INT_TO_UDINT(MINUTE) * UDINT#60 + _INT_TO_UDINT(HOUR) * UDINT#3600;
END_FUNCTION

PROGRAM program0

	VAR
		YEAR :	INT;
		MONTH :	INT;
		DAY :	INT;
		HOUR :	INT;
		MINUTE :	INT;
		SECOND :	INT;
		CEIL5_OUT : UDINT;
	END_VAR

	CEIL5_OUT := SET_DT(YEAR, MONTH, DAY, HOUR, MINUTE, SECOND);

END_PROGRAM

CONFIGURATION Config0

	RESOURCE Res0 ON PLC
		TASK task0(INTERVAL := T#20ms,PRIORITY := 0);
		PROGRAM instance0 WITH task0 : program0;
	END_RESOURCE

END_CONFIGURATION

(* ---- SET_TOD.ST ---- *)
FUNCTION _REAL_TO_UDINT:UDINT

	VAR_INPUT
		X :	REAL;
	END_VAR

	IF REAL_TO_UDINT(0.5) = UDINT#1 THEN
		_REAL_TO_UDINT := REAL_TO_UDINT(x);
	ELSIF X > 0.0 THEN
		_REAL_TO_UDINT := REAL_TO_UDINT(x+0.5);
	ELSIF X < 0.0 THEN
		_REAL_TO_UDINT := REAL_TO_UDINT(x-0.5);
	ELSE
		_REAL_TO_UDINT := UDINT#0;
	END_IF;

END_FUNCTION

FUNCTION _INT_TO_UDINT:UDINT

	VAR_INPUT
		IN :	INT;
	END_VAR

	_INT_TO_UDINT := DINT_TO_UDINT(INT_TO_DINT(IN));

END_FUNCTION

FUNCTION SET_TOD:UDINT

	VAR_INPUT
		HOUR :	INT;
		MINUTE :	INT;
		SECOND :	REAL;
	END_VAR

	set_Tod := _REAL_TO_UDINT(second * 1000.0) + _INT_TO_UDINT(minute) * UDINT#60000 + _INT_TO_UDINT(hour) * UDINT#3600000;

END_FUNCTION

PROGRAM program0

	VAR
		HOUR :	INT;
		MINUTE :	INT;
		SECOND :	REAL;
		CEIL5_OUT : UDINT;
	END_VAR

	CEIL5_OUT := SET_TOD(HOUR, MINUTE, SECOND);

END_PROGRAM

CONFIGURATION Config0

	RESOURCE Res0 ON PLC
		TASK task0(INTERVAL := T#20ms,PRIORITY := 0);
		PROGRAM instance0 WITH task0 : program0;
	END_RESOURCE

END_CONFIGURATION

(* ---- SETUP_EXTENDED_ASCII.ST ---- *)
FUNCTION SETUP_EXTENDED_ASCII:BOOL

	VAR_INPUT
		X :	BOOL;
	END_VAR

	SETUP_EXTENDED_ASCII := X OR TRUE;
END_FUNCTION

PROGRAM program0
  VAR
	X :	BOOL;
    CEIL5_OUT : BOOL;
  END_VAR

  CEIL5_OUT := SETUP_EXTENDED_ASCII(X);
END_PROGRAM

CONFIGURATION Config0

  RESOURCE Res0 ON PLC
    TASK task0(INTERVAL := T#20ms,PRIORITY := 0);
    PROGRAM instance0 WITH task0 : program0;
  END_RESOURCE
END_CONFIGURATION

(* ---- SGN.ST ---- *)
FUNCTION SGN : INT
  VAR_INPUT
    x : REAL;
  END_VAR

  IF X > 0.0 THEN
  	sgn := 1;
  ELSIF X < 0.0 THEN
  	sgn := -1;
  ELSE
  	sgn := 0;
  END_IF;
END_FUNCTION

PROGRAM program0
  VAR
    LocalVar0 : REAL;
    LocalVar1 : INT;
    CEIL5_OUT : INT;
  END_VAR

  CEIL5_OUT := SGN(LocalVar0);
  LocalVar1 := CEIL5_OUT;
END_PROGRAM

CONFIGURATION Config0

  RESOURCE Res0 ON PLC
    TASK task0(INTERVAL := T#20ms,PRIORITY := 0);
    PROGRAM instance0 WITH task0 : program0;
  END_RESOURCE
END_CONFIGURATION

(* ---- SHL1.ST ---- *)
FUNCTION SHL1:DWORD

	VAR_INPUT
		IN :	DWORD;
		N :	INT;
	END_VAR

	SHL1 := SHR(DWORD#16#FF_FF_FF_FF,32-N) OR SHL(IN,N);

END_FUNCTION

PROGRAM program0

	VAR
		IN :	DWORD;
		N :	INT;
		CEIL5_OUT : DWORD;
	END_VAR

  	CEIL5_OUT := SHL1(IN, N);

END_PROGRAM

CONFIGURATION Config0

	RESOURCE Res0 ON PLC
		TASK task0(INTERVAL := T#20ms,PRIORITY := 0);
		PROGRAM instance0 WITH task0 : program0;
	END_RESOURCE

END_CONFIGURATION

(* ---- SHR1.ST ---- *)
FUNCTION SHR1:DWORD

	VAR_INPUT
		IN :	DWORD;
		N :	INT;
	END_VAR

	SHR1 := SHL(DWORD#16#FF_FF_FF_FF,32-N) OR SHR(IN,N);

END_FUNCTION

PROGRAM program0

	VAR
		IN : DWORD;
		N :	INT;
		CEIL5_OUT : DWORD;
	END_VAR

	CEIL5_OUT := SHR1(IN, N);

END_PROGRAM

CONFIGURATION Config0

	RESOURCE Res0 ON PLC
		TASK task0(INTERVAL := T#20ms,PRIORITY := 0);
		PROGRAM instance0 WITH task0 : program0;
	END_RESOURCE

END_CONFIGURATION

(* ---- SIGMOID.ST ---- *)
FUNCTION SIGMOID:REAL

	VAR_INPUT
		X :	REAL;
	END_VAR

	IF X > 20.0 THEN
		SIGMOID := 1.0;
	ELSIF x < -85.0 THEN
		SIGMOID := 0.0;
	ELSE
		SIGMOID := 1.0 / (1.0 + EXP(-X));
	END_IF;

END_FUNCTION

PROGRAM program0

	VAR
		X :	REAL;
		CEIL5_OUT : REAL;
	END_VAR

	CEIL5_OUT := SIGMOID(X);

END_PROGRAM

CONFIGURATION Config0

	RESOURCE Res0 ON PLC
		TASK task0(INTERVAL := T#20ms,PRIORITY := 0);
		PROGRAM instance0 WITH task0 : program0;
	END_RESOURCE

END_CONFIGURATION

(* ---- SIGN_I.ST ---- *)
FUNCTION BIT_OF_DWORD : BOOL

	VAR_INPUT
		IN : DWORD;
		N : INT;
	END_VAR

	BIT_OF_DWORD := (SHR(in,N) AND 16#00000001) > 0;

END_FUNCTION

FUNCTION SIGN_I:BOOL

	VAR_INPUT
		IN :	DINT;
	END_VAR

	sign_I := BIT_OF_DWORD(DINT_TO_DWORD(in),31);

END_FUNCTION

PROGRAM program0

	VAR
		IN :	DINT;
		CEIL5_OUT : BOOL;
	END_VAR

	CEIL5_OUT := SIGN_I(IN);

END_PROGRAM

CONFIGURATION Config0

	RESOURCE Res0 ON PLC
		TASK task0(INTERVAL := T#20ms,PRIORITY := 0);
		PROGRAM instance0 WITH task0 : program0;
	END_RESOURCE

END_CONFIGURATION

(* ---- SIGN_R.ST ---- *)
FUNCTION SIGN_R : BOOL
  VAR_INPUT
    IN : REAL;
  END_VAR

  SIGN_R := in < 0.0;
END_FUNCTION

PROGRAM program0
  VAR
    LocalVar0 : REAL;
    CEIL5_OUT : BOOL;
  END_VAR

  CEIL5_OUT := SIGN_R(LocalVar0);
END_PROGRAM

CONFIGURATION Config0

  RESOURCE Res0 ON PLC
    TASK task0(INTERVAL := T#20ms,PRIORITY := 0);
    PROGRAM instance0 WITH task0 : program0;
  END_RESOURCE
END_CONFIGURATION

(* ---- SINC.ST ---- *)
FUNCTION SINC:REAL

	VAR_INPUT
		X :	REAL;
	END_VAR

	IF X = 0.0 THEN
		SINC := 1.0;
	ELSE
		SINC := SIN(x) / x;
	END_IF;

END_FUNCTION

PROGRAM program0

	VAR
		X :	REAL;
		CEIL5_OUT : REAL;
	END_VAR

  	CEIL5_OUT := SINC(X);

END_PROGRAM

CONFIGURATION Config0

	RESOURCE Res0 ON PLC
		TASK task0(INTERVAL := T#20ms,PRIORITY := 0);
		PROGRAM instance0 WITH task0 : program0;
	END_RESOURCE

END_CONFIGURATION

(* ---- SINH.ST ---- *)
FUNCTION SINH:REAL
	VAR_INPUT
		X :	REAL;
	END_VAR

	IF ABS(x) < 2.0E-3 THEN
		SINH := X;
	ELSE
		SINH := (EXP(x) - EXP(-x)) * 0.5;
	END_IF;
END_FUNCTION

PROGRAM program0
  VAR
    LocalVar0 : REAL;
    CEIL5_OUT : REAL;
  END_VAR

  CEIL5_OUT := SINH(LocalVar0);
END_PROGRAM

CONFIGURATION Config0

  RESOURCE Res0 ON PLC
    TASK task0(INTERVAL := T#20ms,PRIORITY := 0);
    PROGRAM instance0 WITH task0 : program0;
  END_RESOURCE
END_CONFIGURATION

(* ---- SPHERE_V.ST ---- *)
FUNCTION SPHERE_V:REAL

	VAR_INPUT
		RX :	REAL;
	END_VAR

	sphere_V := 4.188790205 * Rx * RX * RX;

END_FUNCTION

PROGRAM program0

	VAR
		RX :	REAL;
		CEIL5_OUT : REAL;
	END_VAR

	CEIL5_OUT := SPHERE_V(RX);

END_PROGRAM

CONFIGURATION Config0

	RESOURCE Res0 ON PLC
		TASK task0(INTERVAL := T#20ms,PRIORITY := 0);
		PROGRAM instance0 WITH task0 : program0;
	END_RESOURCE

END_CONFIGURATION

(* ---- SQRTN.ST ---- *)
FUNCTION SQRTN:REAL

	VAR_INPUT
		X :	REAL;
		N :	INT;
	END_VAR

	IF N > 0 THEN
		SQRTN := EXP(LN(x) / INT_TO_REAL(n));
	ELSE
		SQRTN := 0.0;
	END_IF;

END_FUNCTION

PROGRAM program0
	VAR
		LocalVar0 : REAL;
		LocalVar1 : INT;
		LocalOUT  : REAL;
	END_VAR

 	LocalOUT := SQRTN(LocalVar0, LocalVar1);

END_PROGRAM

CONFIGURATION Config0

	RESOURCE Res0 ON PLC
		TASK task0(INTERVAL := T#20ms,PRIORITY := 0);
		PROGRAM instance0 WITH task0 : program0;
	END_RESOURCE

END_CONFIGURATION

(* ---- STAIR.ST ---- *)
FUNCTION _REAL_TO_DINT:DINT
	VAR_INPUT
		X :	REAL;
	END_VAR

	IF REAL_TO_DINT(0.5) = DINT#1 THEN
		_REAL_TO_DINT := REAL_TO_DINT(x);
		RETURN;
	END_IF;

	IF X > 0.0 THEN
		_REAL_TO_DINT := REAL_TO_DINT(x+0.5);
	ELSIF X < 0.0 THEN
		_REAL_TO_DINT := REAL_TO_DINT(x-0.5);
	ELSE
		_REAL_TO_DINT := DINT#0;
	END_IF;

END_FUNCTION

FUNCTION STAIR:REAL

	VAR_INPUT
		X :	REAL;
		D :	REAL;
	END_VAR

	IF D > 0.0 THEN
		STAIR := DINT_TO_REAL(_REAL_TO_DINT(X / D)) * D;
	ELSE
		STAIR := X;
	END_IF;

END_FUNCTION

PROGRAM program0

	VAR
		X :	REAL;
		D :	REAL;
		CEIL5_OUT : REAL;
	END_VAR

	CEIL5_OUT := STAIR(X, D);

END_PROGRAM

CONFIGURATION Config0

	RESOURCE Res0 ON PLC
		TASK task0(INTERVAL := T#20ms,PRIORITY := 0);
		PROGRAM instance0 WITH task0 : program0;
	END_RESOURCE

END_CONFIGURATION

(* ---- SUN_MIDDAY.ST ---- *)
FUNCTION _REAL_TO_UDINT:UDINT
	VAR_INPUT
		X :	REAL;
	END_VAR

	IF REAL_TO_UDINT(0.5) = UDINT#1 THEN
		_REAL_TO_UDINT := REAL_TO_UDINT(x);
	ELSIF X > 0.0 THEN
		_REAL_TO_UDINT := REAL_TO_UDINT(x+0.5);
	ELSIF X < 0.0 THEN
		_REAL_TO_UDINT := REAL_TO_UDINT(x-0.5);
	ELSE
		_REAL_TO_UDINT := UDINT#0;
	END_IF;

END_FUNCTION

FUNCTION HOUR_TO_TOD:UDINT

	VAR_INPUT
		IN :	REAL;
	END_VAR

	hour_to_tod := _REAL_TO_UDINT(IN * 3600000.00);

END_FUNCTION

FUNCTION DAY_OF_YEAR:INT
	VAR_INPUT
		IDATE :	DATE;
	END_VAR

	DAY_OF_YEAR := UDINT_TO_INT((DATE_TO_UDINT(idate) / UDINT#86400) MOD UDINT#1461);
	IF DAY_OF_YEAR > 729 THEN
		IF DAY_OF_YEAR > 1095 THEN DAY_OF_YEAR := DAY_OF_YEAR - 1095; ELSE DAY_OF_YEAR := DAY_OF_YEAR - 729; END_IF;
	ELSIF DAY_OF_YEAR > 364 THEN
		DAY_OF_YEAR := DAY_OF_YEAR - 364;
	ELSE
		DAY_OF_YEAR := DAY_OF_YEAR + 1;
	END_IF;
END_FUNCTION

FUNCTION SUN_MIDDAY:UDINT

	VAR_INPUT
		LON :	REAL;
		UTC :	DATE;
	END_VAR

	VAR
		T :	REAL;
		OFFSET :	REAL;
	END_VAR

	T := INT_TO_REAL(DAY_OF_YEAR(utc));
	OFFSET := -0.1752 * SIN(0.033430 * T + 0.5474) - 0.1340 * SIN(0.018234 * T - 0.1939);
	SUN_MIDDAY := HOUR_TO_TOD(12.0 - OFFSET - lon * 0.0666666666666);

END_FUNCTION

PROGRAM program0

	VAR
		LON :	REAL;
		UTC :	DATE;
		CEIL5_OUT : UDINT;
	END_VAR

	CEIL5_OUT := SUN_MIDDAY(LON, UTC);

END_PROGRAM

CONFIGURATION Config0

	RESOURCE Res0 ON PLC
		TASK task0(INTERVAL := T#20ms,PRIORITY := 0);
		PROGRAM instance0 WITH task0 : program0;
	END_RESOURCE

END_CONFIGURATION

(* ---- SWAP_BYTE.ST ---- *)
FUNCTION SWAP_BYTE:WORD

	VAR_INPUT
		IN :	WORD;
	END_VAR

	Swap_Byte := ROL(in,8);

END_FUNCTION

PROGRAM program0

	VAR
		IN :	WORD;
		CEIL5_OUT : WORD;
	END_VAR

	CEIL5_OUT := SWAP_BYTE(IN);

END_PROGRAM

CONFIGURATION Config0

	RESOURCE Res0 ON PLC
		TASK task0(INTERVAL := T#20ms,PRIORITY := 0);
		PROGRAM instance0 WITH task0 : program0;
	END_RESOURCE

END_CONFIGURATION

(* ---- SWAP_BYTE2.ST ---- *)
FUNCTION SWAP_BYTE2:DWORD

	VAR_INPUT
		INPUT :	DWORD;
	END_VAR

	Swap_Byte2 := (ROR(INPUT,8) AND DWORD#16#FF00FF00) OR (ROL(INPUT,8) AND DWORD#16#00FF00FF);

END_FUNCTION

PROGRAM program0

	VAR
		IN :	DWORD;
		CEIL5_OUT : DWORD;
	END_VAR

	CEIL5_OUT := SWAP_BYTE2(IN);

END_PROGRAM

CONFIGURATION Config0

	RESOURCE Res0 ON PLC
		TASK task0(INTERVAL := T#20ms,PRIORITY := 0);
		PROGRAM instance0 WITH task0 : program0;
	END_RESOURCE

END_CONFIGURATION

(* ---- TANC.ST ---- *)
FUNCTION TANC:REAL

	VAR_INPUT
		X :	REAL;
	END_VAR

	IF X = 0.0 THEN
		TANC := 1.0;
	ELSE
		TANC := TAN(x) / x;
	END_IF;

END_FUNCTION

PROGRAM program0

	VAR
		X :	REAL;
		CEIL5_OUT : REAL;
	END_VAR

	CEIL5_OUT := TANC(X);

END_PROGRAM

CONFIGURATION Config0

	RESOURCE Res0 ON PLC
		TASK task0(INTERVAL := T#20ms,PRIORITY := 0);
		PROGRAM instance0 WITH task0 : program0;
	END_RESOURCE

END_CONFIGURATION

(* ---- TANH.ST ---- *)
FUNCTION TANH:REAL

	VAR_INPUT
		X :	REAL;
	END_VAR

	IF X > 20.0 THEN
		TANH := 1.0;
	ELSIF X < -20.0 THEN
		TANH := -1.0;
	ELSE
		TANH := 1.0 - 2.0 / (EXP(2.0 * x) + 1.0);
	END_IF;

END_FUNCTION

PROGRAM program0

	VAR
		X :	REAL;
		CEIL5_OUT : REAL;
	END_VAR

	CEIL5_OUT := TANH(X);

END_PROGRAM

CONFIGURATION Config0

	RESOURCE Res0 ON PLC
		TASK task0(INTERVAL := T#20ms,PRIORITY := 0);
		PROGRAM instance0 WITH task0 : program0;
	END_RESOURCE

END_CONFIGURATION

(* ---- TANK_VOL1.ST ---- *)
FUNCTION CIRCLE_SEG:REAL
	VAR_INPUT
		RX :	REAL;
		HX :	REAL;
	END_VAR

	IF RX > 0.0 THEN
		CIRCLE_SEG := 2.0 * ACOS(1.0 - LIMIT(0.0, HX / RX, 2.0));
		CIRCLE_SEG := (CIRCLE_SEG - SIN(CIRCLE_SEG)) * RX * RX * 0.5;
	END_IF;
END_FUNCTION

FUNCTION TANK_VOL1:REAL

	VAR_INPUT
		TR :	REAL;
		TL :	REAL;
		H :	REAL;
	END_VAR

	TANK_VOL1 := CIRCLE_SEG(TR, H) * TL;

END_FUNCTION

PROGRAM program0
  VAR
    TR :	REAL;
	TL :	REAL;
	H :	REAL;
    CEIL5_OUT : REAL;
  END_VAR

  CEIL5_OUT := TANK_VOL1(TR, TL, H);
END_PROGRAM

CONFIGURATION Config0

  RESOURCE Res0 ON PLC
    TASK task0(INTERVAL := T#20ms,PRIORITY := 0);
    PROGRAM instance0 WITH task0 : program0;
  END_RESOURCE
END_CONFIGURATION

(* ---- TANK_VOL2.ST ---- *)
FUNCTION TANK_VOL2:REAL

	VAR_INPUT
		TR :	REAL;
		H :	REAL;
	END_VAR

	TANK_VOL2 := 3.14159265358979323846264338327950288 * H * H * (TR - H / 3.0);

END_FUNCTION

PROGRAM program0
  VAR
    TR :	REAL;
	H :	REAL;
    CEIL5_OUT : REAL;
  END_VAR

  CEIL5_OUT := TANK_VOL2(TR, H);
END_PROGRAM

CONFIGURATION Config0

  RESOURCE Res0 ON PLC
    TASK task0(INTERVAL := T#20ms,PRIORITY := 0);
    PROGRAM instance0 WITH task0 : program0;
  END_RESOURCE
END_CONFIGURATION

(* ---- TEMP_NI.ST ---- *)
FUNCTION TEMP_NI:REAL
	VAR_INPUT
		RES :	REAL;
		R0 :	REAL;
	END_VAR

	TEMP_NI := (SQRT(0.30085225 - 2.66E-3 * (R0 - Res)) - 0.5485) * 751.8796992;
END_FUNCTION

PROGRAM program0
  	VAR
		RES :	REAL;
		R0 :	REAL;
    	CEIL5_OUT : REAL;
  	END_VAR

  	CEIL5_OUT := TEMP_NI(RES, R0);
END_PROGRAM

CONFIGURATION Config0
	RESOURCE Res0 ON PLC
		TASK task0(INTERVAL := T#20ms,PRIORITY := 0);
		PROGRAM instance0 WITH task0 : program0;
	END_RESOURCE
END_CONFIGURATION

(* ---- TEMP_NTC.ST ---- *)
FUNCTION TEMP_NTC:REAL

VAR_INPUT
	RES :	REAL;
	RN :	REAL;
	B :	REAL;
END_VAR

IF res > 0.0 THEN
	TEMP_NTC := B * 298.15 / (B + LN(RES / RN) * 298.15) -273.15;
END_IF;

END_FUNCTION

PROGRAM program0
  	VAR
		RES :	REAL;
		RN :	REAL;
		B :	REAL;
    	CEIL5_OUT : REAL;
  	END_VAR

  	CEIL5_OUT := TEMP_NTC(RES, RN, B);
END_PROGRAM

CONFIGURATION Config0
	RESOURCE Res0 ON PLC
		TASK task0(INTERVAL := T#20ms,PRIORITY := 0);
		PROGRAM instance0 WITH task0 : program0;
	END_RESOURCE
END_CONFIGURATION

(* ---- TEMP_PT.ST ---- *)
FUNCTION RES_PT:REAL
	VAR_INPUT
		T :	REAL;
		R0 :	REAL;
	END_VAR

	VAR
		T2 :	REAL;
	END_VAR

	T2 := T * T;

	IF T >= 0.0 THEN
		RES_PT := R0 * ( 1.0 + 3.90802E-3 * T + -5.802E-7 * T2);
	ELSE
		RES_PT := R0 * ( 1.0 + 3.90802E-3 * T + -5.802E-7 * T2 + -4.27350E-12 * (T - 100.0) * T2 * T);
	END_IF;

END_FUNCTION

FUNCTION TEMP_PT:REAL

	VAR_INPUT
		RES :	REAL;
		R0 :	REAL;
	END_VAR

	VAR
		step_var :	REAL := REAL#50.0;
		X :	REAL;
		Y :	REAL;
		t1 :	REAL;
	END_VAR

	X := 3.9083E-3 * R0;
	Y := -5.775E-7 * R0;
	IF Res >= R0 THEN
		t1 := X * X - 4.0 * Y * (R0 - Res);
		IF t1 < 0.0 THEN
			TEMP_PT := 10000.0;
		ELSE
			TEMP_PT := (-X + SQRT(t1)) / (2.0 * Y);
		END_IF;
	ELSE
		TEMP_PT := -100.0;
		WHILE step_var > 0.01 DO
			IF RES_PT(TEMP_PT, R0) < res THEN TEMP_PT := TEMP_PT + step_var; ELSE TEMP_PT := TEMP_PT - step_var; END_IF;
			step_var := step_var * 0.5;
		END_WHILE;
	END_IF;
END_FUNCTION

PROGRAM program0
	VAR
		RES :	REAL;
		R0 :	REAL;
		CEIL5_OUT : REAL;
	END_VAR

	CEIL5_OUT := TEMP_PT(RES, R0);
END_PROGRAM

CONFIGURATION Config0
	RESOURCE Res0 ON PLC
		TASK task0(INTERVAL := T#20ms,PRIORITY := 0);
		PROGRAM instance0 WITH task0 : program0;
	END_RESOURCE
END_CONFIGURATION

(* ---- TEMP_SI.ST ---- *)
FUNCTION TEMP_SI:REAL
	VAR_INPUT
		RES :	REAL;
		VAR_RS:	REAL;
		TS :	REAL;
	END_VAR

	TEMP_SI := (-7.64E-3 + SQRT(RES/VAR_RS* 6.64E-5 - 0.803E-5)) * 30120.48193 + TS;

END_FUNCTION

PROGRAM program0
  	VAR
		RES :	REAL;
		VAR_RS:	REAL;
		TS :	REAL;
    	CEIL5_OUT : REAL;
  	END_VAR

  	CEIL5_OUT := TEMP_SI(RES, VAR_RS, TS);
END_PROGRAM

CONFIGURATION Config0
	RESOURCE Res0 ON PLC
		TASK task0(INTERVAL := T#20ms,PRIORITY := 0);
		PROGRAM instance0 WITH task0 : program0;
	END_RESOURCE
END_CONFIGURATION

(* ---- TIME_TO_DWORD.ST ---- *)
FUNCTION TIME_TO_DWORD1:DWORD

VAR_INPUT
	X :	TIME;
END_VAR

TIME_TO_DWORD1 := UDINT_TO_DWORD(DINT_TO_UDINT(TIME_TO_DINT(X)));
END_FUNCTION

PROGRAM program0
  VAR
	X :	TIME;
    CEIL5_OUT : DWORD;
  END_VAR

  CEIL5_OUT := TIME_TO_DWORD1(X);
END_PROGRAM

CONFIGURATION Config0

  RESOURCE Res0 ON PLC
    TASK task0(INTERVAL := T#20ms,PRIORITY := 0);
    PROGRAM instance0 WITH task0 : program0;
  END_RESOURCE
END_CONFIGURATION

(* ---- TIME_TO_INT.ST ---- *)
FUNCTION TIME_TO_INT1:INT

VAR_INPUT
	IN :	TIME;
END_VAR

TIME_TO_INT1 := DINT_TO_INT(TIME_TO_DINT(IN));
END_FUNCTION

PROGRAM program0
  VAR
	IN :	TIME;
    CEIL5_OUT : INT;
  END_VAR

  CEIL5_OUT := TIME_TO_INT1(IN);
END_PROGRAM

CONFIGURATION Config0

  RESOURCE Res0 ON PLC
    TASK task0(INTERVAL := T#20ms,PRIORITY := 0);
    PROGRAM instance0 WITH task0 : program0;
  END_RESOURCE
END_CONFIGURATION

(* ---- TIME_TO_REAL.ST ---- *)
FUNCTION TIME_TO_REAL1:REAL

VAR_INPUT
	X :	TIME;
END_VAR

TIME_TO_REAL1 := UDINT_TO_REAL(DINT_TO_UDINT(TIME_TO_DINT(X)));
END_FUNCTION

PROGRAM program0
  VAR
	X :	TIME;
    CEIL5_OUT : REAL;
  END_VAR

  CEIL5_OUT := TIME_TO_REAL1(X);
END_PROGRAM

CONFIGURATION Config0

  RESOURCE Res0 ON PLC
    TASK task0(INTERVAL := T#20ms,PRIORITY := 0);
    PROGRAM instance0 WITH task0 : program0;
  END_RESOURCE
END_CONFIGURATION

(* ---- TIME_TO_TOD.ST ---- *)
FUNCTION TIME_TO_TOD:UDINT

	VAR_INPUT
		IN :	TIME;
	END_VAR

	TIME_TO_TOD := DWORD_TO_UDINT(TIME_TO_DWORD(IN));
END_FUNCTION

PROGRAM program0
  VAR
	IN :	TIME;
    CEIL5_OUT : UDINT;
  END_VAR

  CEIL5_OUT := TIME_TO_TOD(IN);
END_PROGRAM

CONFIGURATION Config0

  RESOURCE Res0 ON PLC
    TASK task0(INTERVAL := T#20ms,PRIORITY := 0);
    PROGRAM instance0 WITH task0 : program0;
  END_RESOURCE
END_CONFIGURATION

(* ---- TIME_TO_UDINT.ST ---- *)
FUNCTION TIME_TO_UDINT2:UDINT
	VAR_INPUT
		X :	TIME;
	END_VAR

	TIME_TO_UDINT2 := DINT_TO_UDINT(TIME_TO_DINT(X));
END_FUNCTION

PROGRAM program0
  VAR
    LocalVar0 : TIME;
    LocalOUT  : UDINT;
  END_VAR

  LocalOUT := TIME_TO_UDINT2(LocalVar0);
END_PROGRAM

CONFIGURATION Config0
    RESOURCE Res0 ON PLC
        TASK task0(INTERVAL := T#20ms,PRIORITY := 0);
        PROGRAM instance0 WITH task0 : program0;
    END_RESOURCE
END_CONFIGURATION

(* ---- TIMECHECK.ST ---- *)
FUNCTION TIMECHECK:BOOL

	VAR_INPUT
		TD :	UDINT;
		START :	UDINT;
		STOP :	UDINT;
	END_VAR

	IF stop < start THEN
		TIMECHECK := start <= TD OR  TD < stop;
	ELSE
		TIMECHECK := start <= TD AND TD < stop;
	END_IF;

END_FUNCTION

PROGRAM program0
  VAR
	TD :	UDINT;
	START :	UDINT;
	STOP :	UDINT;
    CEIL5_OUT : BOOL;
  END_VAR

  CEIL5_OUT := TIMECHECK(TD, START, STOP);
END_PROGRAM

CONFIGURATION Config0

  RESOURCE Res0 ON PLC
    TASK task0(INTERVAL := T#20ms,PRIORITY := 0);
    PROGRAM instance0 WITH task0 : program0;
  END_RESOURCE
END_CONFIGURATION

(* ---- TN_SC_SHADOW_ATTR.ST ---- *)
FUNCTION TN_SC_SHADOW_ATTR:BYTE

	VAR_INPUT
		Iby_ATTR :	BYTE;
	END_VAR

	TN_SC_SHADOW_ATTR := ((Iby_ATTR AND BYTE#2#11110000) OR BYTE#2#00001000);

END_FUNCTION

PROGRAM program0
	VAR
		Iby_ATTR :	BYTE;
		CEIL5_OUT : BYTE;
	END_VAR

  	CEIL5_OUT := TN_SC_SHADOW_ATTR(Iby_ATTR);
END_PROGRAM

CONFIGURATION Config0

  RESOURCE Res0 ON PLC
    TASK task0(INTERVAL := T#20ms,PRIORITY := 0);
    PROGRAM instance0 WITH task0 : program0;
  END_RESOURCE
END_CONFIGURATION

(* ---- TN_SC_XY2_ERROR.ST ---- *)
FUNCTION TN_SC_XY2_ERROR:BOOL

	VAR_INPUT
		X1 :	INT;
		Y1 :	INT;
		X2 :	INT;
		Y2 :	INT;
	END_VAR

	TN_SC_XY2_ERROR := Y1 < 0 OR X1 < 0 OR Y2 < 0 OR X2 < 0 OR Y1 > 23 OR X1 > 79 OR Y2 > 23 OR X2 > 79;

END_FUNCTION

PROGRAM program0
	VAR
		X1 :	INT;
		Y1 :	INT;
		X2 :	INT;
		Y2 :	INT;
		CEIL5_OUT : BOOL;
	END_VAR

  	CEIL5_OUT := TN_SC_XY2_ERROR(X1, Y1, X2, Y2);
END_PROGRAM

CONFIGURATION Config0

  RESOURCE Res0 ON PLC
    TASK task0(INTERVAL := T#20ms,PRIORITY := 0);
    PROGRAM instance0 WITH task0 : program0;
  END_RESOURCE
END_CONFIGURATION

(* ---- TN_SC_XY_ERROR.ST ---- *)
FUNCTION TN_SC_XY_ERROR:BOOL

	VAR_INPUT
		X :	INT;
		Y :	INT;
	END_VAR

	TN_SC_XY_ERROR := Y < 0 OR X < 0 OR Y > 23 OR X > 79;

END_FUNCTION

PROGRAM program0
	VAR
		X :	INT;
		Y :	INT;
		CEIL5_OUT : BOOL;
	END_VAR

  	CEIL5_OUT := TN_SC_XY_ERROR(X, Y);
END_PROGRAM

CONFIGURATION Config0

  RESOURCE Res0 ON PLC
    TASK task0(INTERVAL := T#20ms,PRIORITY := 0);
    PROGRAM instance0 WITH task0 : program0;
  END_RESOURCE
END_CONFIGURATION

(* ---- TO_LOWER.ST ---- *)
FUNCTION SETUP_EXTENDED_ASCII:BOOL

	VAR_INPUT
		X :	BOOL;
	END_VAR

	SETUP_EXTENDED_ASCII := X OR TRUE;
END_FUNCTION

FUNCTION TO_LOWER:BYTE

	VAR_INPUT
		IN :	BYTE;
	END_VAR

	IF in > BYTE#64 AND in < BYTE#91 THEN
	TO_LOWER := in OR BYTE#16#20;
	ELSIF (in > BYTE#191 AND in < BYTE#223) AND in <> BYTE#215 AND SETUP_EXTENDED_ASCII(FALSE) THEN
	TO_LOWER := in OR BYTE#16#20;
	ELSE
	TO_LOWER := in;
	END_IF;

END_FUNCTION

PROGRAM program0
  VAR
	IN :	BYTE;
    CEIL5_OUT : BYTE;
  END_VAR

  CEIL5_OUT := TO_LOWER(IN);
END_PROGRAM

CONFIGURATION Config0

  RESOURCE Res0 ON PLC
    TASK task0(INTERVAL := T#20ms,PRIORITY := 0);
    PROGRAM instance0 WITH task0 : program0;
  END_RESOURCE
END_CONFIGURATION

(* ---- TO_UPPER.ST ---- *)
FUNCTION SETUP_EXTENDED_ASCII:BOOL
	VAR_INPUT
		X :	BOOL;
	END_VAR

	SETUP_EXTENDED_ASCII := X OR TRUE;
END_FUNCTION

FUNCTION TO_UPPER:BYTE

	VAR_INPUT
		IN :	BYTE;
	END_VAR

	IF in > BYTE#96 AND in < BYTE#123 THEN
	TO_UPPER := in AND BYTE#16#DF;
	ELSIF in > BYTE#223 AND in <> BYTE#247 AND in <> BYTE#255 AND SETUP_EXTENDED_ASCII(FALSE) THEN
	TO_UPPER := in AND BYTE#16#DF;
	ELSE
	TO_UPPER := in;
	END_IF;

END_FUNCTION

PROGRAM program0
  VAR
	IN :	BYTE;
    CEIL5_OUT : BYTE;
  END_VAR

  CEIL5_OUT := TO_UPPER(IN);
END_PROGRAM

CONFIGURATION Config0

  RESOURCE Res0 ON PLC
    TASK task0(INTERVAL := T#20ms,PRIORITY := 0);
    PROGRAM instance0 WITH task0 : program0;
  END_RESOURCE
END_CONFIGURATION

(* ---- TOD_TO_REAL.ST ---- *)
FUNCTION TOD_TO_REAL2:REAL
	VAR_INPUT
		IN :	UDINT;
	END_VAR
	TOD_TO_REAL2 := UDINT_TO_REAL(IN);
END_FUNCTION

PROGRAM program0
  VAR
	IN :	UDINT;
    CEIL5_OUT : REAL;
  END_VAR

  CEIL5_OUT := TOD_TO_REAL2(IN);
END_PROGRAM

CONFIGURATION Config0

  RESOURCE Res0 ON PLC
    TASK task0(INTERVAL := T#20ms,PRIORITY := 0);
    PROGRAM instance0 WITH task0 : program0;
  END_RESOURCE
END_CONFIGURATION

(* ---- TOD_TO_TIME.ST ---- *)
FUNCTION TOD_TO_TIME:TIME
	VAR_INPUT
		IN :	UDINT;
	END_VAR

	TOD_TO_TIME := DWORD_TO_TIME(UDINT_TO_DWORD(IN));
END_FUNCTION

PROGRAM program0
  VAR
	IN :	UDINT;
    CEIL5_OUT : TIME;
  END_VAR

  CEIL5_OUT := TOD_TO_TIME(IN);
END_PROGRAM

CONFIGURATION Config0

  RESOURCE Res0 ON PLC
    TASK task0(INTERVAL := T#20ms,PRIORITY := 0);
    PROGRAM instance0 WITH task0 : program0;
  END_RESOURCE
END_CONFIGURATION

(* ---- TRIANGLE_A.ST ---- *)
FUNCTION _REAL_TO_DINT:DINT
  VAR_INPUT
    X :	REAL;
  END_VAR

  IF REAL_TO_DINT(0.5) = DINT#1 THEN
    _REAL_TO_DINT := REAL_TO_DINT(x);
    RETURN;
  END_IF;

  IF X > 0.0 THEN
    _REAL_TO_DINT := REAL_TO_DINT(x+0.5);
  ELSIF X < 0.0 THEN
    _REAL_TO_DINT := REAL_TO_DINT(x-0.5);
  ELSE
    _REAL_TO_DINT := DINT#0;
  END_IF;
END_FUNCTION

FUNCTION FLOOR2:DINT

	VAR_INPUT
		X :	REAL;
	END_VAR

	FLOOR2 := _REAL_TO_DINT(X);
	IF DINT_TO_REAL(FLOOR2) > X THEN
		FLOOR2 := FLOOR2 - DINT#1;
	END_IF;

END_FUNCTION

FUNCTION MODR:REAL

	VAR_INPUT
		IN :	REAL;
		DIVI :	REAL;
	END_VAR

	IF divi = 0.0 THEN
		MODR := 0.0;
	ELSE
		MODR := in - DINT_TO_REAL(FLOOR2(in / divi)) * divi;
	END_IF;

END_FUNCTION

FUNCTION RAD:REAL

	VAR_INPUT
		DEG :	REAL;
	END_VAR

	Rad := modR(0.0174532925199433 * deg , 6.283185307179586476);

END_FUNCTION

FUNCTION TRIANGLE_A:REAL

	VAR_INPUT
		S1 :	REAL;
		A :	REAL;
		S2 :	REAL;
		S3 :	REAL;
	END_VAR

	IF A = 0.0 THEN
		TRIANGLE_A := SQRT((s1+s2+S3) * (s1+s2-S3) * (S2+S3-S1) * (S3+S1-S2)) * 0.25;
	ELSE
		TRIANGLE_A := S1 * S2 * SIN(RAD(A)) * 0.5;
	END_IF;

END_FUNCTION

PROGRAM program0
  VAR
	S1 :	REAL;
	A :	REAL;
	S2 :	REAL;
	S3 :	REAL;
    CEIL5_OUT : REAL;
  END_VAR

  CEIL5_OUT := TRIANGLE_A(S1, A, S2, S3);
END_PROGRAM

CONFIGURATION Config0

  RESOURCE Res0 ON PLC
    TASK task0(INTERVAL := T#20ms,PRIORITY := 0);
    PROGRAM instance0 WITH task0 : program0;
  END_RESOURCE
END_CONFIGURATION

(* ---- TRUNC_REAL.ST ---- *)
FUNCTION TRUNC_REAL:REAL

	VAR_INPUT
		IN :	REAL;
	END_VAR

	TRUNC_REAL := UDINT_TO_REAL(DINT_TO_UDINT(TRUNC(IN)));
END_FUNCTION

PROGRAM program0

	VAR
		IN :	REAL;
		OUT: REAL;
	END_VAR
	OUT := TRUNC_REAL(IN);

END_PROGRAM

CONFIGURATION Config0

	RESOURCE Res0 ON PLC
		TASK task0(INTERVAL := T#20ms,PRIORITY := 0);
		PROGRAM instance0 WITH task0 : program0;
	END_RESOURCE

END_CONFIGURATION

(* ---- TRUNC_UDINT.ST ---- *)
FUNCTION TRUNC_UDINT:UDINT
	VAR_INPUT
		IN :	REAL;
	END_VAR
	TRUNC_UDINT := DINT_TO_UDINT(TRUNC(IN));
END_FUNCTION

PROGRAM program0
	VAR
		LocalVar0 : REAL;
		LocalOUT  : UDINT;
	END_VAR
		LocalOUT := TRUNC_UDINT(LocalVar0);
END_PROGRAM

CONFIGURATION Config0
	RESOURCE Res0 ON PLC
		TASK task0(INTERVAL := T#20ms,PRIORITY := 0);
		PROGRAM instance0 WITH task0 : program0;
	END_RESOURCE
END_CONFIGURATION

(* ---- UDINT_TO_TIME.ST ---- *)
FUNCTION _UDINT_TO_TIME:TIME

	VAR_INPUT
		IN :	UDINT;
	END_VAR

	_UDINT_TO_TIME := DINT_TO_TIME(UDINT_TO_DINT(IN));

END_FUNCTION

PROGRAM program0
  VAR
	  IN :	UDINT;
    CEIL5_OUT : TIME;
  END_VAR

  CEIL5_OUT := _UDINT_TO_TIME(IN);
END_PROGRAM

CONFIGURATION Config0

  RESOURCE Res0 ON PLC
    TASK task0(INTERVAL := T#20ms,PRIORITY := 0);
    PROGRAM instance0 WITH task0 : program0;
  END_RESOURCE
END_CONFIGURATION

(* ---- WCT.ST ---- *)
FUNCTION WCT:REAL

	VAR_INPUT
		T :	REAL;
		V :	REAL;
	END_VAR

	IF V < 5.0 OR T > 10.0 THEN
		WCT := T;
	ELSE
		WCT := 13.12 + 0.6215 * T +(0.3965 * T - 11.37) * EXP(LN(v) * 0.16);
	END_IF;

END_FUNCTION

PROGRAM program0
	VAR
		T :	REAL;
		V :	REAL;
		CEIL5_OUT : REAL;
	END_VAR

  	CEIL5_OUT := WCT(T, V);
END_PROGRAM

CONFIGURATION Config0

  RESOURCE Res0 ON PLC
    TASK task0(INTERVAL := T#20ms,PRIORITY := 0);
    PROGRAM instance0 WITH task0 : program0;
  END_RESOURCE
END_CONFIGURATION

(* ---- WINDOW.ST ---- *)
FUNCTION WINDOW:BOOL
	VAR_INPUT
		LOW :	REAL;
		IN :	REAL;
		HIGH :	REAL;
	END_VAR
	window := (in < high) AND (in > low);

END_FUNCTION

PROGRAM program0
  	VAR
		LOW :	REAL;
		IN :	REAL;
		HIGH :	REAL;
		CEIL5_OUT : BOOL;
	END_VAR

  	CEIL5_OUT := window(LOW, IN, HIGH);
END_PROGRAM

CONFIGURATION Config0
  	RESOURCE Res0 ON PLC
    	TASK task0(INTERVAL := T#20ms,PRIORITY := 0);
    	PROGRAM instance0 WITH task0 : program0;
  	END_RESOURCE
END_CONFIGURATION

(* ---- WINDOW2.ST ---- *)
FUNCTION WINDOW2:BOOL
	VAR_INPUT
		LOW :	REAL;
		IN :	REAL;
		HIGH :	REAL;
	END_VAR
	window2 := (in <= high) AND (in >= low);
END_FUNCTION

PROGRAM program0
  	VAR
		LOW :	REAL;
		IN :	REAL;
		HIGH :	REAL;
		CEIL5_OUT : BOOL;
	END_VAR

  	CEIL5_OUT := window2(LOW, IN, HIGH);
END_PROGRAM

CONFIGURATION Config0
  	RESOURCE Res0 ON PLC
    	TASK task0(INTERVAL := T#20ms,PRIORITY := 0);
    	PROGRAM instance0 WITH task0 : program0;
  	END_RESOURCE
END_CONFIGURATION

(* ---- WORD_OF_BYTE.ST ---- *)
FUNCTION WORD_OF_BYTE:WORD
	VAR_INPUT
		B1 :	BYTE;
		B0 :	BYTE;
	END_VAR
	WORD_OF_BYTE := SHL(BYTE_TO_WORD(B1),8) OR BYTE_TO_WORD(B0);
END_FUNCTION

PROGRAM program0
  	VAR
		B1 :	BYTE;
		B0 :	BYTE;
		CEIL5_OUT : WORD;
	END_VAR

  	CEIL5_OUT := WORD_OF_BYTE(B1, B0);
END_PROGRAM

CONFIGURATION Config0
  	RESOURCE Res0 ON PLC
    	TASK task0(INTERVAL := T#20ms,PRIORITY := 0);
    	PROGRAM instance0 WITH task0 : program0;
  	END_RESOURCE
END_CONFIGURATION

(* ---- WORD_OF_DWORD.ST ---- *)
FUNCTION _BYTE_TO_INT:INT
	VAR_INPUT
		IN :	BYTE;
	END_VAR

	_BYTE_TO_INT := USINT_TO_INT(BYTE_TO_USINT(IN));
END_FUNCTION

FUNCTION WORD_OF_DWORD:WORD
	VAR_INPUT
		IN: DWORD;
		N :	BYTE;
	END_VAR
	WORD_OF_DWORD := DWORD_TO_WORD(SHR(in,_BYTE_TO_INT(SHL(n,4))));
END_FUNCTION

PROGRAM program0
  	VAR
		IN :	DWORD;
		N :	BYTE;
		CEIL5_OUT : WORD;
	  END_VAR

  	CEIL5_OUT := WORD_OF_DWORD(IN, N);
END_PROGRAM

CONFIGURATION Config0
  	RESOURCE Res0 ON PLC
    	TASK task0(INTERVAL := T#20ms,PRIORITY := 0);
    	PROGRAM instance0 WITH task0 : program0;
  	END_RESOURCE
END_CONFIGURATION

(* ---- WORD_TO_RANGE.ST ---- *)
FUNCTION _WORD_TO_REAL:REAL
	VAR_INPUT
		IN :	WORD;
	END_VAR
	_WORD_TO_REAL := UINT_TO_REAL(WORD_TO_UINT(IN));
END_FUNCTION

FUNCTION WORD_TO_RANGE:REAL
	VAR_INPUT
		X :	WORD;
		LOW :	REAL;
		HIGH :	REAL;
	END_VAR
	WORD_TO_RANGE := (high - low) * _WORD_TO_REAL(X) * 0.00001525902189669640 + low;
END_FUNCTION

PROGRAM program0
  	VAR
		X :	WORD;
		LOW :	REAL;
		HIGH :	REAL;
		CEIL5_OUT : REAL;
	  END_VAR

  	CEIL5_OUT := WORD_TO_RANGE(X, LOW, HIGH);
END_PROGRAM

CONFIGURATION Config0
  	RESOURCE Res0 ON PLC
    	TASK task0(INTERVAL := T#20ms,PRIORITY := 0);
    	PROGRAM instance0 WITH task0 : program0;
  	END_RESOURCE
END_CONFIGURATION

(* ---- WORK_WEEK.ST ---- *)
FUNCTION LEAP_YEAR:BOOL

  VAR_INPUT
    YEAR :	INT;
  END_VAR

  IF (year MOD INT#400) = INT#00 THEN
    leap_year := TRUE;
  ELSIF (year MOD INT#100) = INT#00 THEN
    leap_year := FALSE;
  ELSIF (year MOD INT#04) = INT#00 THEN
    leap_year := TRUE;
  ELSE
    leap_year := FALSE;
  END_IF;

END_FUNCTION

FUNCTION DAY_OF_WEEK:INT

	VAR_INPUT
		IDATE :	UDINT;
	END_VAR

	DAY_OF_WEEK := UDINT_TO_INT((idate / UDINT#86400 + UDINT#3) MOD UDINT#7) + INT#01;

END_FUNCTION

FUNCTION YEAR_OF_DATE:INT
	VAR_INPUT
		IDATE :	UDINT;
	END_VAR

	YEAR_OF_DATE := UDINT_TO_INT((idate+UDINT#43200) / UDINT#31557600 + UDINT#1970);
END_FUNCTION

FUNCTION _INT_TO_UDINT:UDINT
	VAR_INPUT
		IN :	INT;
	END_VAR

	_INT_TO_UDINT := DINT_TO_UDINT(INT_TO_DINT(IN));
END_FUNCTION

FUNCTION YEAR_BEGIN:UDINT
	VAR_INPUT
		Y :	INT;
	END_VAR
	year_begin := DWORD_TO_UDINT(SHR(UDINT_TO_DWORD(_INT_TO_UDINT(y) * UDINT#1461 - UDINT#2878169),2))*UDINT#86400;

END_FUNCTION

FUNCTION WORK_WEEK:INT

	VAR_INPUT
		IDATE :	UDINT;
	END_VAR

	VAR
		d1 :	UDINT;
		w1 :	INT;
		ds :	UDINT;
		yr :	INT;
		w31 :	INT;
		w01 :	INT;
		wm :	INT;
	END_VAR

	yr := YEAR_OF_DATE(idate);
	d1 := year_begin(yr);
	w1 := DAY_OF_WEEK(d1);
	IF w1 < 5 THEN
		ds := d1 - _INT_TO_UDINT(w1+6) * UDINT#86400;
	ELSE
		ds := d1 + _INT_TO_UDINT(1-w1) * UDINT#86400;
	END_IF;

	work_week := UDINT_TO_INT((idate - ds) / UDINT#604800);

	IF work_week = 0 THEN
		IF w1 > 1 THEN w31 := w1 - 1; ELSE W31 := 7; END_IF;
		IF leap_year(yr - 1) THEN IF w31 > 1 THEN w01 := W31 - 1; ELSE w1 := 7; END_IF; END_IF;
		WORK_WEEK := 52 + BOOL_TO_INT(w31 = 4 OR w01 = 4);
	ELSE
		IF leap_year(yr) THEN
			IF w1 < 7 THEN w31 := w1 + 1; ELSE w31 := 1; END_IF;
		ELSE
			w31 := w1;
		END_IF;
		wm := 52 + BOOL_TO_INT(w31 = 4 OR w1 = 4);
		IF work_week > wm THEN work_week := 1; END_IF;
	END_IF;

END_FUNCTION

PROGRAM program0
  VAR
    Y : UDINT;
    CEIL5_OUT : INT;
  END_VAR

  CEIL5_OUT := WORK_WEEK(Y);
END_PROGRAM

CONFIGURATION Config0

  RESOURCE Res0 ON PLC
    TASK task0(INTERVAL := T#20ms,PRIORITY := 0);
    PROGRAM instance0 WITH task0 : program0;
  END_RESOURCE
END_CONFIGURATION

(* ---- YEAR_BEGIN.ST ---- *)
FUNCTION _INT_TO_UDINT:UDINT
	VAR_INPUT
		IN :	INT;
	END_VAR

	_INT_TO_UDINT := DINT_TO_UDINT(INT_TO_DINT(IN));
END_FUNCTION

FUNCTION YEAR_BEGIN:UDINT
	VAR_INPUT
		Y :	INT;
	END_VAR
	year_begin := DWORD_TO_UDINT(SHR(UDINT_TO_DWORD(_INT_TO_UDINT(y) * UDINT#1461 - UDINT#2878169),2))*UDINT#86400;

END_FUNCTION

PROGRAM program0
  VAR
    Y : INT;
    CEIL5_OUT : UDINT;
  END_VAR

  CEIL5_OUT := YEAR_BEGIN(Y);
END_PROGRAM

CONFIGURATION Config0

  RESOURCE Res0 ON PLC
    TASK task0(INTERVAL := T#20ms,PRIORITY := 0);
    PROGRAM instance0 WITH task0 : program0;
  END_RESOURCE
END_CONFIGURATION

(* ---- YEAR_END.ST ---- *)
FUNCTION YEAR_END:UDINT

	VAR_INPUT
		Y :	INT;
	END_VAR

	YEAR_END := DWORD_TO_UDINT(SHR(UDINT_TO_DWORD(INT_TO_UDINT(y) * UDINT#1461 - UDINT#2876712), 2)) * UDINT#86400;

END_FUNCTION

PROGRAM program0
  VAR
    Y : INT;
    CEIL5_OUT : UDINT;
  END_VAR

  CEIL5_OUT := YEAR_END(Y);
END_PROGRAM

CONFIGURATION Config0

  RESOURCE Res0 ON PLC
    TASK task0(INTERVAL := T#20ms,PRIORITY := 0);
    PROGRAM instance0 WITH task0 : program0;
  END_RESOURCE
END_CONFIGURATION

(* ---- YEAR_OF_DATE.ST ---- *)
FUNCTION YEAR_OF_DATE:INT
	VAR_INPUT
		IDATE :	UDINT;
	END_VAR

	YEAR_OF_DATE := UDINT_TO_INT((idate+UDINT#43200) / UDINT#31557600 + UDINT#1970);
END_FUNCTION

PROGRAM program0
  VAR
    LocalVar0 : UDINT;
    CEIL5_OUT : INT;
  END_VAR

  CEIL5_OUT := YEAR_OF_DATE(LocalVar0);
END_PROGRAM

CONFIGURATION Config0

  RESOURCE Res0 ON PLC
    TASK task0(INTERVAL := T#20ms,PRIORITY := 0);
    PROGRAM instance0 WITH task0 : program0;
  END_RESOURCE
END_CONFIGURATION
